FUNCTION_BLOCK MoveVelocityTestSuite EXTENDS TestSuite<TestSuiteParameter.MaxTestCount>
VAR
END_VAR

END_FUNCTION_BLOCK

(* stored: Version 1.1.0.1
   POU MoveVelocityTestSuite: Id {6f423009-7ac9-4bbc-9784-ede5e34ea635}, SpecialFunc None *)
